{attribute 'linkalways'}
{attribute 'hide_all_locals'}
FUNCTION_BLOCK ValueUdint EXTENDS ValueUdintRead IMPLEMENTS Value
VAR
END_VAR

METHOD SetFromType : BOOL
VAR_INPUT
	source : __SYSTEM.AnyType;
END_VAR
SetFromType := ConvertAnyType(source, thisAnyType);
END_METHOD

METHOD SetFromString : BOOL
VAR_INPUT
	value : T_MaxString;
END_VAR
thisValue := STRING_TO_UDINT(value);

SetFromString := TRUE;
END_METHOD

METHOD Set : BOOL
VAR_INPUT
	source : ANY;
END_VAR
Set := ConvertAnyType(source, thisAnyType);
END_METHOD

END_FUNCTION_BLOCK

(* stored: Version 1.1.0.1
   POU ValueUdint: Id {a113a914-6f98-495c-aee5-22630206bc75}, SpecialFunc None
   Method SetFromType: Id {06032852-dcde-4c5b-afd4-9d3cb6829e84}
   Method SetFromString: Id {d03693bd-395e-4185-8013-f3d8da8e7773}
   Method Set: Id {e95143c3-4b85-4b1d-b178-7440be4d0a3c} *)
